SYSTEM Test Rendezvous
  (* Version 1.0, 2005-11-20, Goran Cengic, Chalmers *)
  DEVICE Test Device : DeviceType_not_used
    RESOURCE Test Resource : ResourceType_not_used
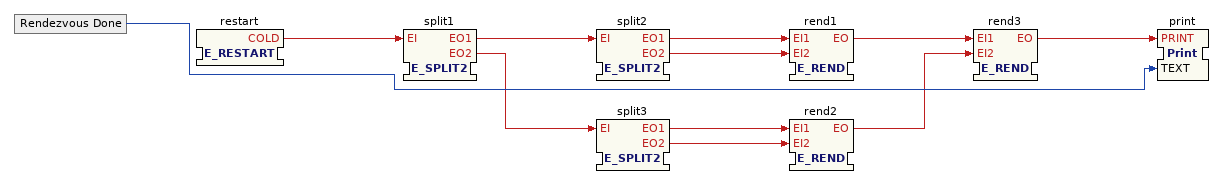
      FBS
        restart : E_RESTART;
        split1 : E_SPLIT2;
        split2 : E_SPLIT2;
        split3 : E_SPLIT2;
        rend1 : E_REND;
        rend2 : E_REND;
        rend3 : E_REND;
        print : Print;
      END_FBS
      EVENT_CONNECTIONS
        restart.COLD TO split1.EI;
        split1.EO1 TO split2.EI;
        split1.EO2 TO split3.EI;
        split2.EO1 TO rend1.EI1;
        split2.EO2 TO rend1.EI2;
        split3.EO1 TO rend2.EI1;
        split3.EO2 TO rend2.EI2;
        rend1.EO TO rend3.EI1;
        rend2.EO TO rend3.EI2;
        rend3.EO TO print.PRINT;
      END_CONNECTIONS
      DATA_CONNECTIONS
        Rendezvous Done TO print.TEXT;
      END_CONNECTIONS
    END_RESOURCE
  END_DEVICE
END_SYSTEM
